// TIA Portal V20 export
DATA_BLOCK "Config"   // DB107
// stored: Access Published, MemoryReserve 100, Namespace Unit1.Em4
   VAR
      em : "LAF_typeEmConfiguration";   // Configuration of EM Parameters
      axis : Array[1.._.U1EM4_NO_OF_AXES] of DB_ANY;
      cam : Array[1.._.U1EM4_NO_OF_AXES] of DB_ANY;
      OutputCam : Array[1.._.U1EM4_NO_OF_AXES] of DB_ANY;
      MeasuringInput : Array[1.._.U1EM4_NO_OF_AXES] of DB_ANY;
      moduleAccessPoint : Array[1.._.U1EM4_NO_OF_AXES] of HW_SUBMODULE;
   END_VAR
   VAR RETAIN
      cmCompensatorAxisZ : "LBC_typeAxisControlConfiguration";
      cmFeedingRollAxisB : "LBC_typeAxisControlConfiguration";
      cmElectrodeCutterAxisZ : "LBC_typeAxisControlConfiguration";
      cmPositionMovingAxisX : "LBC_typeAxis64PosConfiguration";
      cmFeederCylinderUpDown : "LBC_typeTwoWayActuatorConfiguration";
      cmCompensatorSafetyPinIdlePosition : "LBC_typeDigitalSignalConfiguration";
      cmTabDetectSensor : "LBC_typeDigitalSignalConfiguration";
      cmTapeDetectSensor : "LBC_typeDigitalSignalConfiguration";
      cmCutterEpcAnalogInput : "LBC_typeAnalogInputConfiguration";
      cmCompensatorAxisZ_TorqueCal : "LER_typeServoTorqueCalConfigruation";
      cmFeedingRollAxisB_TorqueCal : "LER_typeServoTorqueCalConfigruation";
      cmElectrodeCutterAxisZ_TorqueCal : "LER_typeServoTorqueCalConfigruation";
      cmPositionMovingAxisX_TorqueCal : "LER_typeServoTorqueCalConfigruation";
   END_VAR
BEGIN
   // axis[1] : cmCompensatorAxisZ
   // axis[2] : cmFeedingRollAxisB
   // axis[3] : cmElectrodeCutterAxisZ
   // axis[4] : cmPositionMovingAxisX
   // cam[1] : cmCompensatorAxisZ
   // cam[2] : cmFeedingRollAxisB
   // cam[3] : cmElectrodeCutterAxisZ
   // cam[4] : cmPositionMovingAxisX
   // OutputCam[1] : cmCompensatorAxisZ
   // OutputCam[2] : cmFeedingRollAxisB
   // OutputCam[3] : cmElectrodeCutterAxisZ
   // OutputCam[4] : cmPositionMovingAxisX
   // MeasuringInput[1] : MeasuringInput_FeedingRollAxisB_Tab
   // MeasuringInput[2] : MeasuringInput_FeedingRollAxisB_Tape
   // moduleAccessPoint[1] : cmCompensatorAxisZ
   // moduleAccessPoint[2] : cmFeedingRollAxisB
   // moduleAccessPoint[3] : cmElectrodeCutterAxisZ
   // moduleAccessPoint[4] : cmPositionMovingAxisX
   cmCutterEpcAnalogInput.limitHigh2 := 100.0;
END_DATA_BLOCK
